DATA_BLOCK "Temp_DB"
{ S7_Optimized_Access := 'FALSE' }
VERSION : 0.1
NON_RETAIN
   VAR
      Ana_Temp : Array[1..40] of "UDT_Ana_Temp";   // 模拟量临时变量数组[1..40]

      Device_Temp : Array[1..10] of "UDT_Device_Temp";   // 设备控制临时变量数组[1..10]

      Valve_Temp : Array[1..15] of "UDT_Valve_Temp";   // 阀门控制临时变量数组[1..15]
   END_VAR


BEGIN
END_DATA_BLOCK